FUNCTION_BLOCK FB_TurbVentvalve_NO
VAR_IN_OUT
	iq_stValve : ST_VCC_NO;
END_VAR
VAR_INPUT
	i_stPTM	: ST_AgilentPTM;
END_VAR
VAR
	tofTmr 		: 	TOF;
END_VAR

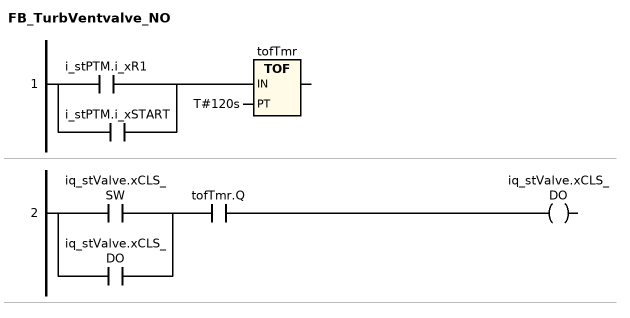
// NETWORK 1
tofTmr(IN := i_stPTM.i_xR1 OR i_stPTM.i_xSTART, PT := T#120s); // TOF

// NETWORK 2
iq_stValve.xCLS_DO := (iq_stValve.xCLS_SW OR iq_stValve.xCLS_DO) AND tofTmr.Q;

END_FUNCTION_BLOCK

(* stored: Version 1.1.0.1, ProductVersion 3.1.4020.12
   POU FB_TurbVentvalve_NO: Id {13f6dcdf-6eaf-4953-b8b2-2ecf46768828}, SpecialFunc None *)
